FUNCTION_BLOCK Detector (* Template for a Basic Function Block Type *)
  (* Standard: 61499-2 *)
  (* Version 1.0, 2023-01-18, obotnar *)
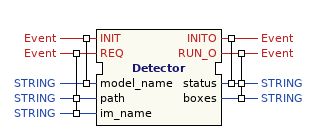
  EVENT_INPUT
    INIT WITH model_name; (* Initialization Request *)
    REQ WITH path, im_name; (* Normal Execution Request *)
  END_EVENT
  EVENT_OUTPUT
    INITO WITH status; (* Initialization Confirm *)
    RUN_O WITH boxes, status; (* Execution Confirmation *)
  END_EVENT
  VAR_INPUT
    model_name : STRING; (* Input event qualifier *)
    path : STRING;
    im_name : STRING;
  END_VAR
  VAR_OUTPUT
    status : STRING; (* Output event qualifier *)
    boxes : STRING;
  END_VAR
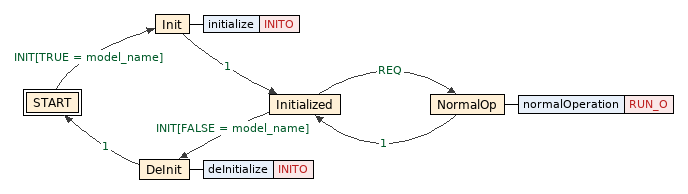
  EC_STATES
    START; (* Initial State *)
    Init : initialize -> INITO; (* Initialization *)
    NormalOp : normalOperation -> RUN_O; (* Normal execution *)
    Initialized;
    DeInit : deInitialize -> INITO;
  END_STATES
  EC_TRANSITIONS
    START TO Init := INIT[TRUE = model_name];
    Init TO Initialized := 1;
    Initialized TO NormalOp := REQ;
    NormalOp TO Initialized := 1;
    DeInit TO START := 1;
    Initialized TO DeInit := INIT[FALSE = model_name];
  END_TRANSITIONS
  ALGORITHM initialize IN ST: (* Initialization algorithm *)
QO := QI;
  END_ALGORITHM
  ALGORITHM deInitialize IN ST: (* Normally executed algorithm *)
QO := FALSE;
  END_ALGORITHM
  ALGORITHM normalOperation IN ST: (* new algorithm *)
QO := QI;

IF TRUE  = QI THEN
  (*  only perform normal operation of QI is true*)

END_IF;
  END_ALGORITHM
END_FUNCTION_BLOCK
